TYPE Std900FastAttenuationConfig EXTENDS DeviceConfiguration :
STRUCT
END_STRUCT
END_TYPE

(* stored: Version 1.1.0.1, ProductVersion 3.1.4024.4
   DUT Std900FastAttenuationConfig: Id {435f9b50-c062-4b41-a77c-099b146b3531} *)
